ABB RobotStudio station: EJERCICIO 3 RESULTO.rspag

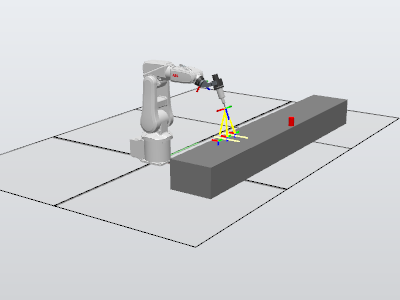
--- station ---
Station mesa-paletizadora2026 (saved by RobotStudio 24.3.10885.0)
Controller IRB120_3_58
  mechanical unit ROB_1: IRB120_3_58__01, 6 joints, base frame (0, 0, 0) mm
Layout (positions relative to the parent item):
  - IRB120_3_58__01 [mechanism, from %ABB.RobotStudio.Models.IRB120%\IRB120_3_58_G_01.rslib] at (0, 0, 0) mm; joint values [0, 0, 0, 0, 0.5236, 0] (rad or m)
  - MyTool [mechanism, from Training Objects\myTool.rslib] at (364.35, 0, 594) mm, rotated rx 180 ry 60 rz 180 deg
  - fotocelulas [smart component]
      signals: DO CajaEn2, DO CajaEn1
      connections:
        LineSensor_2.SensorOut -> fotocelulas.CajaEn2
        LineSensor.SensorOut -> fotocelulas.CajaEn1
    - LineSensor [smart component, from Components\LineSensor.rslib]
        properties: Start=[0.4 0.2 0.215]; End=[0.6 0.2 0.215]; Length=0.2; Radius=0; Tag=(none); SenseMultiple=false; SensedPart=(none); SensedPoint=[0 0 0]
      - _sensorPart_ [part], size 200 x 0 x 0 mm
    - LineSensor_2 [smart component, from Components\LineSensor.rslib]
        properties: Start=[0.4 0.1 0.215]; End=[0.6 0.1 0.215]; Length=0.2; Radius=0; Tag=(none); SenseMultiple=false; SensedPart=(none); SensedPoint=[0 0 0]
      - _sensorPart_ [part], size 200 x 0 x 0 mm
  - CAJA1 [smart component]
      signals: DI Sacar_caja, DI habilitar, DI ventosa, DO colision, DI CAJAen1
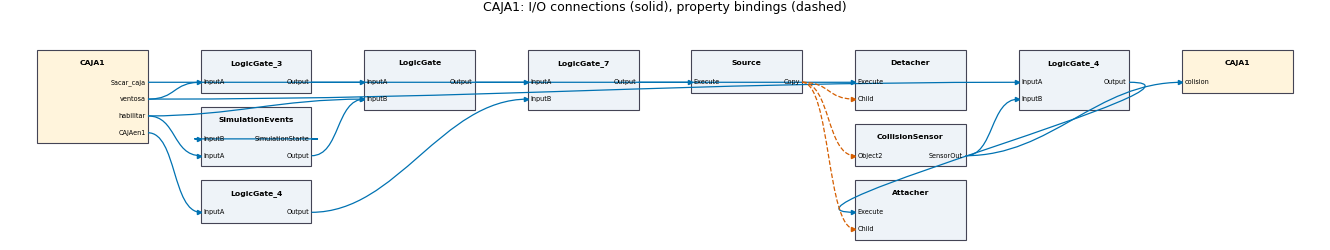
      connections:
        CAJA1.Sacar_caja -> LogicGate.InputA
        LogicGate_3.Output -> Detacher.Execute
        CAJA1.ventosa -> LogicGate_3.InputA
        CollisionSensor.SensorOut -> CAJA1.colision
        CAJA1.ventosa -> LogicGate_4.InputA
        CollisionSensor.SensorOut -> LogicGate_4.InputB
        LogicGate_4.Output -> Attacher.Execute
        SimulationEvents.SimulationStarted -> LogicGate_6.InputB
        CAJA1.habilitar -> LogicGate_2.InputA
        LogicGate_2.Output -> LogicGate.InputB
        CAJA1.habilitar -> LogicGate.InputB
        CAJA1.CAJAen1 -> LogicGate_4.InputA
        LogicGate.Output -> LogicGate_7.InputA
        LogicGate_4.Output -> LogicGate_7.InputB
        LogicGate_7.Output -> Source.Execute
        Source.Copy => Attacher.Child
        Source.Copy => Detacher.Child
        Source.Copy => CollisionSensor.Object2
    - Source [smart component, from Components\Source.rslib]
        properties: Source=caja; Copy=(none); Parent=(none); Position=[0.5 0.2 0.2]; Orientation=[0 0 0]; Transient=true; PhysicsBehavior=3
    - LogicGate [smart component, from Components\LogicGate.rslib]
        properties: Operator=AND; Delay=0
    - Attacher [smart component, from Components\Attacher.rslib]
        properties: Parent=MyTool; Flange=0; Child=(none); Mount=false; Offset=[0 0 0]; Orientation=[0 0 0]
    - Detacher [smart component, from Components\Detacher.rslib]
        properties: Child=(none); KeepPosition=true
    - LogicGate_3 [smart component, from Components\LogicGate.rslib]
        properties: Operator=NOT; Delay=0
    - CollisionSensor [smart component, from Components\CollisionSensor.rslib]
        properties: Object1=MyTool; Object2=(none); NearMiss=0.002; Part1=SpintecTool; Part2=Link6; CollisionType=2
      - _sensorPart_ [part]
    - LogicGate_4 [smart component, from Components\LogicGate.rslib]
        properties: Operator=AND; Delay=0
    - caja [part], size 50.8 x 40.5 x 30.9 mm
    - LogicGate_3 [smart component, from Components\LogicGate.rslib]
        properties: Operator=NOT; Delay=0
    - LogicGate_4 [smart component, from Components\LogicGate.rslib]
        properties: Operator=NOT; Delay=0
    - LogicGate_7 [smart component, from Components\LogicGate.rslib]
        properties: Operator=AND; Delay=0
  - baliza [smart component]
      signals: DI encender
      connections:
        baliza.encender -> Highlighter.Active
    - baliza [part] at (100, 400, 0) mm, size 41 x 41 x 61 mm
    - Highlighter [smart component, from Components\Highlighter.rslib]
        properties: Object=baliza; Color=[0 255 0]; Opacity=255
  - CAJA2 [smart component]
      signals: DI Sacar_caja2, DI habilitar2, DI ventosa2, DO colision2, DI cajaEn2
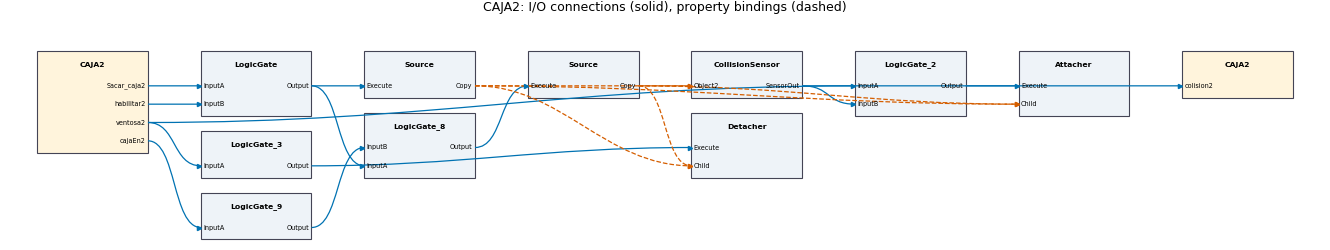
      connections:
        CAJA2.Sacar_caja2 -> LogicGate.InputA
        CAJA2.habilitar2 -> LogicGate.InputB
        LogicGate.Output -> Source.Execute
        CAJA2.ventosa2 -> LogicGate_2.InputA
        CollisionSensor.SensorOut -> LogicGate_2.InputB
        LogicGate_2.Output -> Attacher.Execute
        CAJA2.ventosa2 -> LogicGate_3.InputA
        LogicGate_3.Output -> Detacher.Execute
        CollisionSensor.SensorOut -> CAJA2.colision2
        CAJA2.cajaEn2 -> LogicGate_9.InputA
        LogicGate_9.Output -> LogicGate_8.InputB
        LogicGate.Output -> LogicGate_8.InputA
        LogicGate_8.Output -> Source.Execute
        Source.Copy => CollisionSensor.Object2
        Source.Copy => Detacher.Child
        Source.Copy => Attacher.Child
        Source.Copy => Attacher.Child
        Source.Copy => Detacher.Child
        Source.Copy => CollisionSensor.Object2
    - LogicGate [smart component, from Components\LogicGate.rslib]
        properties: Operator=AND; Delay=0
    - LogicGate_2 [smart component, from Components\LogicGate.rslib]
        properties: Operator=AND; Delay=0
    - Attacher [smart component, from Components\Attacher.rslib]
        properties: Parent=MyTool; Flange=0; Child=(none); Mount=false; Offset=[0 0 0]; Orientation=[0 0 0]
    - Detacher [smart component, from Components\Detacher.rslib]
        properties: Child=(none); KeepPosition=true
    - CollisionSensor [smart component, from Components\CollisionSensor.rslib]
        properties: Object1=MyTool; Object2=(none); NearMiss=0; Part1=SpintecTool; Part2=Link6; CollisionType=2
      - _sensorPart_ [part]
    - LogicGate_3 [smart component, from Components\LogicGate.rslib] at (0, -300, 0) mm
        properties: Operator=NOT; Delay=0
    - caja_2 [part], size 50.8 x 40.5 x 30.9 mm
    - Source [smart component, from Components\Source.rslib]
        properties: Source=caja_2; Copy=(none); Parent=(none); Position=[0.5 0.1 0.2]; Orientation=[0 0 0]; Transient=true; PhysicsBehavior=3
    - LogicGate_8 [smart component, from Components\LogicGate.rslib]
        properties: Operator=AND; Delay=0
    - LogicGate_9 [smart component, from Components\LogicGate.rslib]
        properties: Operator=NOT; Delay=0
  - LogicGate [smart component, from Components\LogicGate.rslib]
      properties: Operator=OR; Delay=0
  - SmartComponent_1 [smart component]
      signals: DI mover_mesa
      connections:
        SmartComponent_1.mover_mesa -> LinearMover2_2.Execute
    - Pieza_1 [part] at (550, 600, 0) mm, size 308.4 x 2009.3 x 205.6 mm
    - LinearMover2_2 [smart component, from Components\LinearMover2.rslib]
        properties: Object=Pieza_1; Direction=[0 -0.001 0]; Distance=0.04; Duration=1; Reference=Global; ReferenceObject=(none)
Attachment: MyTool is attached to IRB120_3_58__01 / Link6
Station signals: DO habilitar, DO ventosa, DO cajaEn1, DO CajaEn2, DI SACAR_CAJA1, DI SACAR_CAJA2, DI TERMINAR_PROCESO, DI STOP_RUN
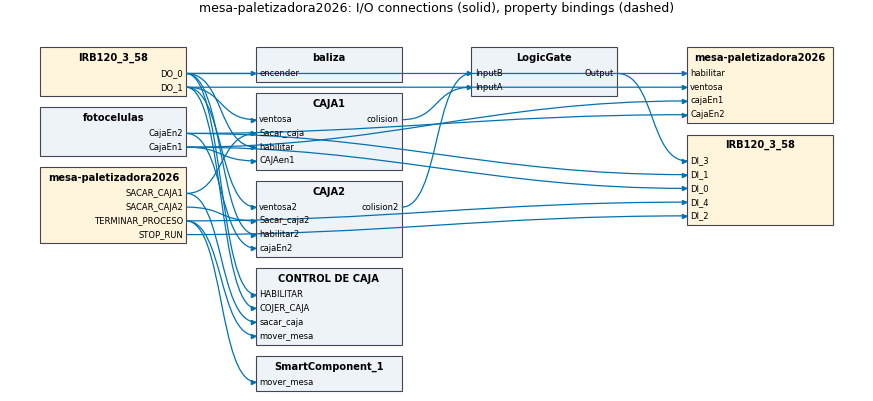
Station logic (signal -> signal, property => property):
  IRB120_3_58.DO_0 -> CONTROL DE CAJA.HABILITAR
  IRB120_3_58.DO_1 -> CONTROL DE CAJA.COJER_CAJA
  IRB120_3_58.DO_0 -> mesa-paletizadora2026.habilitar
  IRB120_3_58.DO_1 -> mesa-paletizadora2026.ventosa
  IRB120_3_58.DO_1 -> CAJA1.ventosa
  IRB120_3_58.DO_0 -> baliza.encender
  IRB120_3_58.DO_1 -> CAJA2.ventosa2
  CAJA2.colision2 -> LogicGate.InputB
  CAJA1.colision -> LogicGate.InputA
  LogicGate.Output -> IRB120_3_58.DI_3
  fotocelulas.CajaEn2 -> IRB120_3_58.DI_1
  fotocelulas.CajaEn1 -> IRB120_3_58.DI_0
  fotocelulas.CajaEn1 -> mesa-paletizadora2026.cajaEn1
  fotocelulas.CajaEn2 -> mesa-paletizadora2026.CajaEn2
  mesa-paletizadora2026.SACAR_CAJA1 -> ?.sacar_caja
  mesa-paletizadora2026.SACAR_CAJA1 -> CAJA1.Sacar_caja
  mesa-paletizadora2026.SACAR_CAJA2 -> CAJA2.Sacar_caja2
  IRB120_3_58.DO_0 -> CAJA2.habilitar2
  IRB120_3_58.DO_0 -> CAJA1.habilitar
  fotocelulas.CajaEn1 -> CAJA1.CAJAen1
  fotocelulas.CajaEn2 -> CAJA2.cajaEn2
  mesa-paletizadora2026.TERMINAR_PROCESO -> IRB120_3_58.DI_4
  mesa-paletizadora2026.TERMINAR_PROCESO -> ?.mover_mesa
  mesa-paletizadora2026.TERMINAR_PROCESO -> SmartComponent_1.mover_mesa
  mesa-paletizadora2026.STOP_RUN -> IRB120_3_58.DI_2

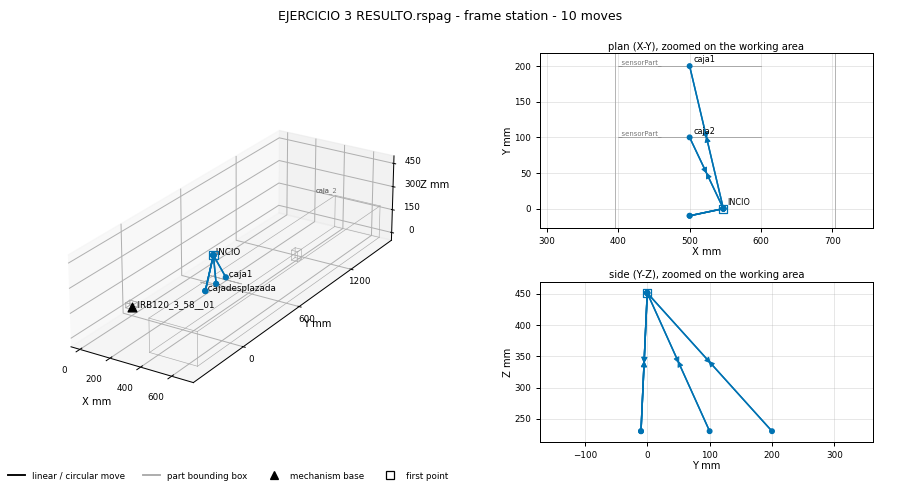
[picture p0: tool path of EJERCICIO 3 RESULTO.rspag in frame station, 10 of 10 moves have a stored position in this frame; points joined in program order, loops and branches not executed]
--- Controller Data/IRB120_3_58/RAPID/TASK1/PROGMOD/CalibData.mod ---
MODULE CalibData
    PERS tooldata MyTool:=[TRUE,[[31.7926,0,229.639],[0.945519,0,0.325568,0]],[1,[0,0,1],[1,0,0,0],0,0,0]];
    TASK PERS wobjdata Workobject_1:=[FALSE,TRUE,"",[[0,0,0],[1,0,0,0]],[[0,0,0],[1,0,0,0]]];
ENDMODULE

--- Controller Data/IRB120_3_58/RAPID/TASK1/PROGMOD/Module1.mod ---
MODULE Module1

    CONST robtarget INCIO:=[[547.330736772,0,451.647300748],[0.190809274,0,0.981627129,0],[0,0,0,0],[9E+09,9E+09,9E+09,9E+09,9E+09,9E+09]];
    CONST robtarget caja1:=[[500.000005126,200.000011571,229.999983554],[0.000000011,0.000000003,1,0.000000012],[0,-1,0,0],[9E+09,9E+09,9E+09,9E+09,9E+09,9E+09]];
    CONST robtarget caja2:=[[500.000004241,100.000005775,229.999972217],[0.000000005,-0.000000006,1,-0.000000001],[0,-1,0,0],[9E+09,9E+09,9E+09,9E+09,9E+09,9E+09]];
    CONST robtarget cajadesplazada:=[[500.000000582,-10.000000181,229.999974246],[-0.000000003,0,1,0],[-1,0,-1,0],[9E+09,9E+09,9E+09,9E+09,9E+09,9E+09]];

!ENTRADAS
!DI_0   SENSOR EN CAJA 1  caja situada en 500,200,200
!DI_1   SENSOR EN CAJA 2  caja situada en 500,100,200
!DI_2   STOP/RUN.   STOP a 0,  RUN a 1
!DI_3   no utilizada
!DI_4   PULSADOR TRABAJO TERMINADO

!SALIDAS
!DO_0  BALIZA
!DO_1 VENTOSA
!DO_0  luz verde DO_0 a 1,  luz roja, DO_0 a 0

    PROC main()

        TPErase;
        SET DO_0;
        TPErase;
          TPWrite "Coloca una pieza";
          WAITTIME 4;
            IF di_0=0 AND di_1=0 THEN
           TPWrite "SIN PIEZA EN LA MESA";
           WAITTIME 2;
            ENDIF
        IF di_0=1 AND di_2=1 THEN
            TPERASE;

        TPErase;
        RESET DO_0;
        ENDIF
        IF DI_0=1 THEN
            RESET DO_0;
            MoveL INCIO,v1000,z100,MyTool\WObj:=wobj0;
              MoveLDO caja1,v1000,z0,MyTool\WObj:=wobj0,DO_1,1;
               MoveL INCIO,v1000,z100,MyTool\WObj:=wobj0;
                MoveL cajadesplazada,v500,z100,MyTool\WObj:=Workobject_1;
                WaitTime 2;
                Reset DO_1;
                 MoveL INCIO,v1000,z100,MyTool\WObj:=wobj0;
                  TPWrite "Pulsa terminar proceso";
       WaitDI DI_4,1;

        ENDIF
        IF DI_1=1 AND di_2=1 THEN
            RESET DO_0;
            MoveL INCIO,v1000,z100,MyTool\WObj:=wobj0;
              MoveLDO caja2,v1000,z0,MyTool\WObj:=wobj0,DO_1,1;
               MoveL INCIO,v1000,z100,MyTool\WObj:=wobj0;
                MoveL cajadesplazada,v500,z100,MyTool\WObj:=Workobject_1;
                WaitTime 2;
                Reset DO_1;
                 MoveL INCIO,v1000,z100,MyTool\WObj:=wobj0;
                    TPWrite "Pulsa terminar proceso";
       WaitDI DI_4,1;

        ENDIF






    ENDPROC

ENDMODULE

--- Controller Data/IRB120_3_58/SYSPAR/EIO.cfg ---
EIO:CFG_1.0:6:1::
#
INDUSTRIAL_NETWORK:

      -Name "DeviceNet" -Label "DeviceNet Master/Slave Network" -Address "2"
#
DEVICENET_DEVICE:

      -Name "d652" -VendorName "ABB Robotics" -ProductName "24 VDC I/O Device"\
      -Label "DSQC 652 24 VDC I/O Device" -Address 10 -ProductCode 26\
      -DeviceType 7 -ConnectionType "COS" -OutputSize 2 -InputSize 2
#
DEVICENET_INTERNAL_DEVICE:

      -Name "DN_Internal_Device" -VendorName "ABB Robotics"\
      -ProductName "DeviceNet Internal Slave Device"
#
EIO_SIGNAL:

      -Name "DI_0" -SignalType "DI" -Device "d652" -DeviceMap "0" -Access "All"

      -Name "DI_1" -SignalType "DI" -Device "d652" -DeviceMap "1" -Access "All"

      -Name "DI_2" -SignalType "DI" -Device "d652" -DeviceMap "2" -Access "All"

      -Name "DI_3" -SignalType "DI" -Device "d652" -DeviceMap "3" -Access "All"

      -Name "DI_4" -SignalType "DI" -Device "d652" -DeviceMap "4" -Access "All"

      -Name "DI_5" -SignalType "DI" -Device "d652" -DeviceMap "5" -Access "All"

      -Name "DO_0" -SignalType "DO" -Device "d652" -DeviceMap "0" -Access "All"

      -Name "DO_1" -SignalType "DO" -Device "d652" -DeviceMap "1" -Access "All"

      -Name "DO_2" -SignalType "DO" -Device "d652" -DeviceMap "2" -Access "All"

      -Name "DO_3" -SignalType "DO" -Device "d652" -DeviceMap "3" -Access "All"

      -Name "DO_4" -SignalType "DO" -Device "d652" -DeviceMap "4" -Access "All"

      -Name "DO_5" -SignalType "DO" -Device "d652" -DeviceMap "5" -Access "All"
